FUNCTION_BLOCK AllEMeters
VAR_INPUT
END_VAR
VAR_OUTPUT
END_VAR
VAR
	OneEnergyMeter: Lib.OneEnergyMeter;
	
	EMeter_A : OneEnergyMeter;
	EMeter_B : OneEnergyMeter;
	
END_VAR

Lib.GVL.nInputCoilIndex      := Lib.GVL_DataHalls.StartInputCoilIndex_E_Meter;
Lib.GVL.nOutputCoilIndex     := Lib.GVL_DataHalls.StartOutputCoilIndex_E_Meter;
Lib.GVL.nInputRegisterIndex  := Lib.GVL_DataHalls.StartInputRegisterIndex_E_Meter;
Lib.GVL.nOutputRegisterIndex := Lib.GVL_DataHalls.StartOutputRegisterIndex_E_Meter;




EMeter_A(
	Status:= Lib.GVL_Em.EM[1].Status, 
	Operating_Hrs:= Lib.GVL_Em.EM[1].Operating_Hrs, 
	Energy:= Lib.GVL_Em.EM[1].Energy, 
	Volume:= Lib.GVL_Em.EM[1].Volume, 
	Supply_Temp:= Lib.GVL_Em.EM[1].Supply_Temp, 
	Return_Temp:= Lib.GVL_Em.EM[1].Return_Temp, 
	Temp_Diff:= Lib.GVL_Em.EM[1].Temp_Diff, 
	Offline:= Lib.GVL_DECI.Term31Offline OR Lib.GVL_Em.EM[1].CommsError
	);
	
EMeter_B(
	Status:= Lib.GVL_Em.EM[2].Status, 
	Operating_Hrs:= Lib.GVL_Em.EM[2].Operating_Hrs, 
	Energy:= Lib.GVL_Em.EM[2].Energy, 
	Volume:= Lib.GVL_Em.EM[2].Volume, 
	Supply_Temp:= Lib.GVL_Em.EM[2].Supply_Temp, 
	Return_Temp:= Lib.GVL_Em.EM[2].Return_Temp, 
	Temp_Diff:= Lib.GVL_Em.EM[2].Temp_Diff, 
	Offline:= Lib.GVL_DECI.Term31Offline OR Lib.GVL_Em.EM[2].CommsError
	);

END_FUNCTION_BLOCK

(* stored: Version 1.1.0.1, ProductVersion 3.1.4024.12
   POU AllEMeters: Id {0513168b-19f2-48d7-b2be-f3a9640ca40b}, SpecialFunc None *)
